FUNCTION_BLOCK FB_Comm_MQTT_Influx EXTENDS FB_Comm_MQTT
VAR_INPUT
END_VAR
VAR_OUTPUT
END_VAR
VAR
	RaDec		: ST_RaDecCoordinate := (RightAscension := GVL_Math.LREAL_MIN, Declination := GVL_Math.LREAL_MIN);
	AltAz		: ST_AltAzCoordinate := (Altitude := GVL_Math.LREAL_MIN, Azimuth := GVL_Math.LREAL_MIN);
	dropped		: INT := 0;	// lines too long for the 255 character buffer, not published
	deliveryFailed	: INT := 0;	// fbMqttClient.Publish() returned FALSE (e.g. client busy/not connected); periodic telemetry, not retried on purpose (#5)
	// 0.0 doubles as "no data received yet" and FB_CO_REFRACT's own "estimate from altitude"
	// sentinel, so a consumer can pass these straight through with no guard needed.
	Temperature	: LREAL := 0.0;	// last received ambient temperature (deg C), set via MQTT by an external weather-station bridge
	Humidity	: LREAL := GVL_Math.LREAL_MIN;	// last received relative humidity (%); unconsumed anywhere today
	Pressure	: LREAL := 0.0;	// last received atmospheric pressure (hPa)

	// revert Temperature/Pressure to their safe defaults if nothing fresh arrives for a while,
	// instead of serving an arbitrarily stale weather reading forever
	bWeatherMessageReceived	: BOOL;
	tonWeatherStale			: TON := (PT := T#10M);
END_VAR

SUPER^();

tonWeatherStale(IN := NOT bWeatherMessageReceived, PT := T#10M);
bWeatherMessageReceived := FALSE;
IF tonWeatherStale.Q THEN
	Temperature := 0.0;
	Pressure := 0.0;
END_IF

METHOD _handleMQTTMessage : BOOL
VAR_INPUT
	sPayloadRcv		: STRING(255);
END_VAR
// A message can carry several parameter=value pairs (command a=1,b=2). Data fields (rightascension, declination,
// elevation, azimuth, ...) are applied first and track/slew last, so they always use the coordinates of this
// message, whatever the field order; for a single-field message nothing changes (BROTLib#39).
_DispatchPass(sPayloadRcv := sPayloadRcv, bVerbPass := FALSE);
_DispatchPass(sPayloadRcv := sPayloadRcv, bVerbPass := TRUE);
END_METHOD

// Runs one parameter=value pair of a 'command' message. Same dispatch as before the multi-field change (BROTLib#39).
METHOD PRIVATE _ApplyField
VAR_INPUT
	parameter		: STRING(255);
	value			: STRING(255);
	sPayloadRcv		: STRING(255);	// the whole payload, only for the log messages
END_VAR
IF parameter = 'power' AND Telescope <> 0 THEN
	// there is no power-off command: Park() serves that role
	IF STRING_TO_UINT(value) = 1 THEN
		Telescope.CoverAutoOpen := TRUE;
		Telescope.Init();
	ELSIF STRING_TO_UINT(value) = 2 THEN
		Telescope.CoverAutoOpen := FALSE;
		Telescope.Init();
	ELSE
		ADSLOGSTR( ADSLOG_MSGTYPE_WARN OR ADSLOG_MSGTYPE_LOG, 'MQTT power: unrecognized value (want 1 or 2) %s', sPayloadRcv);
	END_IF
ELSIF parameter = 'park' AND Telescope <> 0 THEN
	Telescope.Park();
ELSIF parameter = 'gohome' AND Telescope <> 0 THEN
	Telescope.Home();
ELSIF parameter = 'track' AND Telescope <> 0 THEN
	// rightascension/declination are buffered here: they arrive either as separate messages beforehand (pyBROT,
	// BROTgui today) or in the same message as track (the data pass in _DispatchPass runs first, BROTLib#39);
	// an incomplete pair is dropped with a log entry
	IF RaDec.RightAscension > GVL_Math.LREAL_MIN AND RaDec.Declination > GVL_Math.LREAL_MIN THEN
		Telescope.Track(RaDec.RightAscension, RaDec.Declination);
	ELSE
		ADSLOGSTR( ADSLOG_MSGTYPE_WARN OR ADSLOG_MSGTYPE_LOG, 'MQTT track: rightascension/declination incomplete, command dropped %s', sPayloadRcv);
	END_IF
	RaDec.RightAscension := GVL_Math.LREAL_MIN;
	RaDec.Declination := GVL_Math.LREAL_MIN;
ELSIF parameter = 'slew' AND Telescope <> 0 THEN
	// see 'track' above -- same buffer-and-consume pattern, same incomplete-pair gap
	IF AltAz.Azimuth > GVL_Math.LREAL_MIN AND AltAz.Altitude > GVL_Math.LREAL_MIN THEN
		Telescope.Slew(AltAz.Azimuth, AltAz.Altitude);
	ELSE
		ADSLOGSTR( ADSLOG_MSGTYPE_WARN OR ADSLOG_MSGTYPE_LOG, 'MQTT slew: azimuth/elevation incomplete, command dropped %s', sPayloadRcv);
	END_IF
	AltAz.Azimuth := GVL_Math.LREAL_MIN;
	AltAz.Altitude := GVL_Math.LREAL_MIN;
ELSIF parameter = 'stop' AND Telescope <> 0 THEN
	Telescope.Stop();
ELSIF parameter = 'reset' AND Telescope <> 0 THEN
	Telescope.Reset();
ELSIF parameter = 'nasmyth' AND Nasmyth <> 0 THEN
	Nasmyth.SetNasmyth(STRING_TO_USINT(value));
ELSIF parameter = 'rightascension' THEN
	RaDec.RightAscension := STRING_TO_LREAL(value);
ELSIF parameter = 'declination' THEN
	RaDec.Declination := STRING_TO_LREAL(value);
ELSIF parameter = 'elevation' THEN
	AltAz.Altitude := STRING_TO_LREAL(value);
ELSIF parameter = 'azimuth' THEN
	AltAz.Azimuth := STRING_TO_LREAL(value);
ELSIF parameter = 'temperature' THEN
	Temperature := STRING_TO_LREAL(value);
	bWeatherMessageReceived := TRUE;
ELSIF parameter = 'humidity' THEN
	Humidity := STRING_TO_LREAL(value);
	bWeatherMessageReceived := TRUE;
ELSIF parameter = 'pressure' THEN
	Pressure := STRING_TO_LREAL(value);
	bWeatherMessageReceived := TRUE;
ELSIF parameter = 'dut1' AND AltAzTelescope <> 0 THEN
	AltAzTelescope.Dut1 := STRING_TO_LREAL(value);
ELSIF parameter = 'focus' AND Focus <> 0 THEN
	Focus.Position := STRING_TO_LREAL(value);
ELSIF parameter = 'cover_open' AND MirrorCovers <> 0 THEN
	MirrorCovers.Open();
ELSIF parameter = 'cover_close' AND MirrorCovers <> 0 THEN
	MirrorCovers.Close();	
ELSIF parameter = 'dome_open' THEN
	IF Dome <> 0 THEN
		Dome.Open();
	ELSIF Roof <> 0 THEN
		Roof.Open();
	END_IF
ELSIF parameter = 'dome_close' THEN
	IF Dome <> 0 THEN
		Dome.Close();
	ELSIF Roof <> 0 THEN
		Roof.Close();
	END_IF
ELSIF parameter = 'dome_stop' AND (Dome <> 0 OR Roof <> 0) THEN
	IF Dome <> 0 THEN
		Dome.Stop();
	ELSIF Roof <> 0 THEN
		Roof.Stop();
	END_IF		
ELSIF parameter = 'dome_park' AND Dome <> 0 THEN
	Dome.Park();
ELSIF parameter = 'dome_track' AND Dome <> 0 THEN
	IF value = '1'THEN
		Dome.Track();
	ELSE
		Dome.StopTrack();
	END_IF	
ELSIF parameter = 'dome_reset' AND Dome <> 0 THEN
	Dome.Reset();
ELSIF parameter = 'filter' AND Filter <> 0 THEN
	Filter.SetFilter(STRING_TO_USINT(value));
ELSIF (parameter = 'derotator' OR parameter = 'derotatoroffset') AND AltAzTelescope <> 0 THEN
	// two client-facing names for the same thing -- I_AltAzTelescope only has one derotator
	// property (DerotatorOffset), there's no separate "absolute derotator position" concept
	AltAzTelescope.DerotatorOffset := STRING_TO_LREAL(value);
ELSIF parameter = 'elevationoffset' AND AltAzTelescope <> 0 THEN
	AltAzTelescope.AltitudeOffset := STRING_TO_LREAL(value);
ELSIF parameter = 'azimuthoffset' AND AltAzTelescope <> 0 THEN
	AltAzTelescope.AzimuthOffset := STRING_TO_LREAL(value);
ELSIF parameter = 'declinationoffset' AND RaDecTelescope <> 0 THEN
	RaDecTelescope.DeclinationOffset := STRING_TO_LREAL(value);
ELSIF parameter = 'hourangleoffset' AND RaDecTelescope <> 0 THEN
	RaDecTelescope.HourAngleOffset := STRING_TO_LREAL(value);
ELSE
	ADSLOGSTR( ADSLOG_MSGTYPE_WARN OR ADSLOG_MSGTYPE_LOG, 'MQTT not understood %s', sPayloadRcv);
END_IF
END_METHOD

// Walks the parameter=value pairs of a payload via FB_InfluxMessage.remaining and applies the ones that belong to
// this pass: bVerbPass FALSE applies everything except track/slew, TRUE applies only track/slew. Running the
// data pass first means track/slew always see the coordinates of the SAME message (any field order), and a
// single-field message behaves exactly as before. At most MAX_FIELDS pairs are walked per message.
METHOD PRIVATE _DispatchPass
VAR_INPUT
	sPayloadRcv		: STRING(255);
	bVerbPass		: BOOL;
END_VAR
VAR
	influxMessage	: FB_InfluxMessage;
	sNext			: STRING(255);
	nFields			: INT;
	bVerb			: BOOL;
END_VAR
VAR CONSTANT
	MAX_FIELDS		: INT := 8;
END_VAR
sNext := sPayloadRcv;
WHILE sNext <> '' AND nFields < MAX_FIELDS DO
	nFields := nFields + 1;
	influxMessage(sPayload := sNext);
	IF influxMessage.measurement <> 'command' THEN
		RETURN;
	END_IF
	bVerb := influxMessage.parameter = 'track' OR influxMessage.parameter = 'slew';
	IF bVerb = bVerbPass THEN
		_ApplyField(parameter := influxMessage.parameter, value := influxMessage.value, sPayloadRcv := sPayloadRcv);
	END_IF
	sNext := influxMessage.remaining;
END_WHILE
IF sNext <> '' AND NOT bVerbPass THEN
	ADSLOGSTR( ADSLOG_MSGTYPE_WARN OR ADSLOG_MSGTYPE_LOG, 'MQTT more than 8 fields in one message, the rest is ignored %s', sPayloadRcv);
END_IF
END_METHOD

METHOD Publish : BOOL
VAR_INPUT
	domain			: STRING(255) := 'environment';
	location		: STRING(255) := 'roof';
	parameter		: STRING(255);
	value			: STRING(255);
END_VAR
VAR_OUTPUT
	published	: BOOL;
END_VAR
VAR
	sPayloadPub		: STRING(255) := '';
	fbFormat		: FB_FormatString;
	bError			: BOOL;
	nErrID			: UDINT;
	retain_message	: BOOL := FALSE;
	bIsBool			: BOOL;
	sDomain			: STRING(255);
	sLocation		: STRING(255);
	sHost			: STRING(255);
	sKey			: STRING(255);
	sFieldVal		: STRING(255);
	sTopic			: STRING(255);
	sTimestamp		: STRING(20);
	sFormat			: STRING(40);
END_VAR
//sPayloadPub := 'environment,location=roof,host=CX-4E6032 ';
// tag values and the field key are escaped (a space or comma in the host name would break the line); the field
// value is typed by F_InfluxFieldValue: integer 'i', float, boolean or quoted string
sDomain := F_EscapeInfluxTag(domain, FALSE);
sLocation := F_EscapeInfluxTag(location, TRUE);
sHost := F_EscapeInfluxTag(HostName, TRUE);
sKey := F_EscapeInfluxTag(parameter, TRUE);
sFieldVal := F_InfluxFieldValue(value);

// retain message if value is boolean: booleans are meant to be published on change only, so a subscriber that
// connects later gets the current state from the broker
bIsBool := (value = 'TRUE') OR (value = 'FALSE') OR (value = 'true') OR (value = 'false');
retain_message := bIsBool;

// a retained line carries the time it was published, so a replay after a Telegraf restart is stored at that time
// and not at the time of the replay (#38). Consumers must accept the optional timestamp (pyBROT#40).
sTimestamp := '';
IF retain_message THEN
	sTimestamp := F_InfluxTimestamp(F_GetSystemTime());
END_IF
IF sTimestamp <> '' THEN
	sFormat := '%s,location=%s,host=%s %s=%s %s';
ELSE
	sFormat := '%s,location=%s,host=%s %s=%s';
END_IF

fbFormat(
	sFormat 	:= sFormat,
	arg1 		:= F_STRING(sDomain),
	arg2 		:= F_STRING(sLocation),
	arg3 		:= F_STRING(sHost),
	arg4 		:= F_STRING(sKey),
	arg5 		:= F_STRING(sFieldVal),
	arg6 		:= F_STRING(sTimestamp),
	sOut 		=> sPayloadPub,
	bError 		=> bError,
	nErrID 		=> nErrID
);

// a line that did not fit the buffer is cut off and would be invalid (or wrong): do not publish it
IF bError OR LEN(sPayloadPub) >= 255 THEN
	published := FALSE;
	IF dropped < 32767 THEN
		dropped := dropped + 1;
	END_IF
	IF dropped = 1 OR (dropped MOD 100) = 0 THEN
		ADSLOGSTR(ADSLOG_MSGTYPE_WARN OR ADSLOG_MSGTYPE_LOG, 'Influx line too long, not published: %s', parameter);
	END_IF
	Publish := published;
	RETURN;
END_IF

// publish under a per-subsystem sub-topic (domain is already the Influx measurement, e.g.
// 'telescope'/'power'/'electronics'/'hydraulics'/'diagnostics') so a consumer that only cares
// about one subsystem can subscribe to just that sub-topic instead of the whole site's firehose
sTopic := CONCAT(CONCAT(sTopicPublish, '/'), domain);

// bQueue left FALSE on purpose: this is periodic telemetry (republished every 1-5s or on the
// static-fields timer), so a dropped publish under load is self-healing next cycle -- queuing
// would just build a backlog of stale values behind whatever caused the client to be busy.
// One-time events (PublishLog) get bQueue := TRUE instead, see there. (#5)
published := fbMqttClient.Publish(
	sTopic			:= sTopic,
	pPayload		:= ADR(sPayloadPub),
	nPayloadSize	:= LEN2(ADR(sPayloadPub)),
	eQoS			:= TcIotMqttQos.AtMostOnceDelivery,
	bRetain			:= retain_message,
	bQueue			:= FALSE
);

IF NOT published THEN
	IF deliveryFailed < 32767 THEN
		deliveryFailed := deliveryFailed + 1;
	END_IF
	IF deliveryFailed = 1 OR (deliveryFailed MOD 100) = 0 THEN
		ADSLOGSTR(ADSLOG_MSGTYPE_WARN OR ADSLOG_MSGTYPE_LOG, 'MQTT publish failed (client busy/not connected): %s', parameter);
	END_IF
END_IF

Publish := published;
END_METHOD

METHOD PublishLog : BOOL
VAR_INPUT
	level		: STRING(255) := 'INFO';
	message		: STRING(255);
END_VAR
VAR
	sPayloadPub		: STRING(255) := '';
	fbFormat		: FB_FormatString;
	bError			: BOOL;
	nErrID			: UDINT;
	sEscapedMessage	: STRING(255);
	sHost			: STRING(255);
	sLevel			: STRING(255);
	nMaxMessage		: INT;
END_VAR
VAR_OUTPUT
	published	: BOOL;
END_VAR
//sPayloadPub := 'environment,location=roof,host=CX-4E6032 ';
sHost := F_EscapeInfluxTag(HostName, TRUE);
sLevel := F_EscapeInfluxTag(level, TRUE);
sEscapedMessage := F_EscapeInfluxString(message);

// a long message is shortened so that the line fits the 255 character buffer and its closing quote is kept:
// 255 minus 'log,host=' (9), ',level=' (7), ' message="' (10) and the closing '"' (1)
nMaxMessage := 255 - 27 - LEN(sHost) - LEN(sLevel);
sEscapedMessage := F_TruncateInfluxEscaped(sEscapedMessage, nMaxMessage);

fbFormat(
	sFormat := 'log,host=%s,level=%s message="%s"',
	arg1 	:= F_STRING(sHost),
	arg2 	:= F_STRING(sLevel),
	arg3 	:= F_STRING(sEscapedMessage),
	sOut 	=> sPayloadPub,
	bError 	=> bError,
	nErrID 	=> nErrID
);

// still too long (very long host name or level): publish nothing rather than a broken line
IF bError OR LEN(sPayloadPub) >= 255 THEN
	published := FALSE;
	PublishLog := published;
	RETURN;
END_IF

// bQueue TRUE: unlike Publish()'s periodic telemetry, a log/event message is one-time -- if the
// client can't send it immediately, queue it for retry instead of losing it silently (#5)
published := fbMqttClient.Publish(
	sTopic			:= sTopicLog,
	pPayload		:= ADR(sPayloadPub),
	nPayloadSize	:= LEN2(ADR(sPayloadPub)),
	eQoS			:= TcIotMqttQos.AtMostOnceDelivery,
	bRetain			:= FALSE,
	bQueue			:= TRUE
);

PublishLog := published;
END_METHOD

END_FUNCTION_BLOCK

(* stored: Version 1.1.0.1, ProductVersion 3.1.4024.15
   POU FB_Comm_MQTT_Influx: Id {48590b1c-8149-4a75-a4a7-086285ed3fbf}, SpecialFunc None
   Method _handleMQTTMessage: Id {6b8170c3-1db8-4027-aca0-99823e943d46}
   Method _ApplyField: Id {b1996a41-13ee-4523-87f0-a3610dac6f65}
   Method _DispatchPass: Id {7e928bbe-332a-4f98-8267-b812825faa63}
   Method Publish: Id {0b9304dc-7cd5-4e61-ac34-34dd3afe6924}
   Method PublishLog: Id {dd46de85-b82a-4d9d-9238-d6c509f88651} *)
